// TIA Portal V18 export
DATA_BLOCK "RollerV3_DB"   // DB10
VERSION : 0.1
// stored: AutoNumber true, DBAccessibleFromOPCUA true, InstanceOfName RollerV3, InstanceOfType FB
"RollerV3"
   // VAR_INPUT
   //    "E-STOP" : Bool;
   //    SystemON : Bool;
   //    Mode : Int;
   //    SetSpeed : Real;
   //    DirectionLeftRight : Bool;
   //    Offsetspeed : DInt;
   //    YAxisVelocity : DInt;
   //    Roller_HW_address : HW_HSC;
   //    DoorSensors : Bool;
   // END_VAR
   // VAR_OUTPUT
   //    WebDBRollerOutput : Bool;
   //    RollerDirection : Bool;
   //    RollerLinearVelocity : DInt;
   //    RollerRPM : Real;
   //    RollerRPM_Measured : Real;
   // END_VAR
   // VAR_IN_OUT
   //    WebDBStart : Bool;
   //    WebDBStop : Bool;
   // END_VAR
   // VAR
   //    RollerSetReset : Bool;
   //    RollerFullPower : Bool;
   //    RollerHalfPower : Bool;
   //    RollerActive : Bool;
   //    RollerSpeedInputGeneral { ExternalAccessible := 'False'; ExternalVisible := 'False'; ExternalWritable := 'False'} : Real;
   //    RollerSpeedInputPID : Real;
   //    RollerManualValue : Int;
   //    Direction_Plus { ExternalAccessible := 'False'; ExternalVisible := 'False'; ExternalWritable := 'False'} : Bool;
   //    Direction_Minus { ExternalAccessible := 'False'; ExternalVisible := 'False'; ExternalWritable := 'False'} : Bool;
   //    PulseSignalMeasurement : DWord;
   //    MaintenanceM3DirDis : Bool;
   //    MaintenanceSkipPID : Bool;
   //    MaintenanceAutomaticDifVel : Bool;
   //    MaintenanceRollerON : Bool;
   //    RollerDirectionInt_last : Int;
   //    Roller_RPM_Send_last : Real;
   //    RollerSetReset_M : Bool;
   //    RollerSetReset_M2 : Bool;
   //    hscData : HSC_Period;
   // END_VAR
BEGIN
END_DATA_BLOCK
